TYPE PT1T2_Parameter_Strukt :
STRUCT
	K :			REAL;
	T1 :		REAL;
	T2 :		REAL;
END_STRUCT
END_TYPE

(* stored: Version 1.1.0.1, ProductVersion 3.1.4024.13
   DUT PT1T2_Parameter_Strukt: Id {f6fb54f0-0c2e-47dd-90a6-f98ba3602b97} *)
